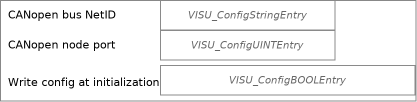
VISUALIZATION VISU_FaulhaberDriveConfig_General  // 417x102
VAR_IN_OUT
	active : FaulhaberDriveConfig;
	editable : FaulhaberDriveConfig;
END_VAR
    Label (5,0 125x30), "CANopen bus NetID"
    Frame (160,0 175x30)
        shows VISU_ConfigStringEntry(active := active.CANopenBusNetId, editable := editable.CANopenBusNetId)
    Label (5,30 125x30), "CANopen node port"
    Frame (160,30 175x30)
        shows VISU_ConfigUINTEntry(active := active.CANopenNodePort, editable := editable.CANopenNodePort)
    Frame (160,65 255x30)
        shows VISU_ConfigBOOLEntry(active := active.sendAtInitialization, editable := editable.sendAtInitialization)
    Label (5,65 155x35), "Write config at initialization"
END_VISUALIZATION

(* stored: Version 1.1.0.1, ProductVersion 3.1.4019.2
   Visu VISU_FaulhaberDriveConfig_General: Id {5de33f36-3877-4e9a-a19d-1b05cd8f5465} *)
